Staubli VAL3: getFrame.pgx

public program getFrame(string& x_sFrm (dimensions=1))
begin
  x_sFrm=sFrameName

end
